// TIA Portal V19 export
FUNCTION_BLOCK "TYPIC_C105_IF_UPS"   // FB23, FBD
TITLE = TYPIC_C105_IF_UPS: No Break
{ S7_Optimized_Access := 'TRUE' }
AUTHOR : OCOTECH
FAMILY : Typical
NAME : C105.701
// Logisch Object Besturing: C105.601
// 
// De interne functie UPS verzorgt de bewaking van een Noobreak installatie.
// stored: MemoryReserve 10, SetENOAutomatically false
   VAR_INPUT
      IN_STS { ExternalAccessible := 'False'; ExternalVisible := 'False'; ExternalWritable := 'False'} : Bool;   // Status van UPS (Batterij / Werking / Bypass)
      IN_TYD { ExternalAccessible := 'False'; ExternalVisible := 'False'; ExternalWritable := 'False'} : Time;   // Resterende autonomietijd (min)
      IN_PWR { ExternalAccessible := 'False'; ExternalVisible := 'False'; ExternalWritable := 'False'} : Real;   // Resterend vermogen
      IN_SPA1 { ExternalAccessible := 'False'; ExternalVisible := 'False'; ExternalWritable := 'False'} : Real;   // Uitgangsspanning 1
      IN_SPA2 { ExternalAccessible := 'False'; ExternalVisible := 'False'; ExternalWritable := 'False'} : Real;   // Uitgangsspanning 2
      IN_SPA3 { ExternalAccessible := 'False'; ExternalVisible := 'False'; ExternalWritable := 'False'} : Real;   // Uitgangsspanning 3
      IN_STR1 { ExternalAccessible := 'False'; ExternalVisible := 'False'; ExternalWritable := 'False'} : Real;   // Uitgangsstroom 1
      IN_STR2 { ExternalAccessible := 'False'; ExternalVisible := 'False'; ExternalWritable := 'False'} : Real;   // Uitgangsstroom 2
      IN_STR3 { ExternalAccessible := 'False'; ExternalVisible := 'False'; ExternalWritable := 'False'} : Real;   // Uitgangsstroom 3
   END_VAR
   VAR_OUTPUT
      VAR_IF_UPS { ExternalAccessible := 'False'; ExternalVisible := 'False'; ExternalWritable := 'False'} : "C105_VAR_IF_UPS_TYPIC";   // Struct met alle variabelen naar bovenliggende functies
   END_VAR
   VAR
      STO { ExternalWritable := 'False'} : Struct   // Storingen
         A001 { ExternalAccessible := 'False'; ExternalVisible := 'False'} : Bool;   // No Break installatie in bypass
         A002 { ExternalAccessible := 'False'; ExternalVisible := 'False'} : Bool;   // No Break installatie uit bedrijf
      END_STRUCT;
      VAR { ExternalWritable := 'False'} : Struct   // Variabelen
         STS1 { ExternalAccessible := 'False'; ExternalVisible := 'False'} : Bool;   // Status UPS [In batterijwerking]
         STS2 { ExternalAccessible := 'False'; ExternalVisible := 'False'} : Bool;   // Status UPS [In bypass]
         STS3 { ExternalAccessible := 'False'; ExternalVisible := 'False'} : Bool;   // Status UPS [In normale werking]
         TYD { ExternalAccessible := 'False'; ExternalVisible := 'False'} : Time;   // Resterende autonomietijd [min]
         PWR { ExternalAccessible := 'False'; ExternalVisible := 'False'} : Real;   // Resterend vermogen
         SPA1 { ExternalAccessible := 'False'; ExternalVisible := 'False'} : Real;   // Uitgangsspanning 1
         SPA2 { ExternalAccessible := 'False'; ExternalVisible := 'False'} : Real;   // Uitgangsspanning 2
         SPA3 { ExternalAccessible := 'False'; ExternalVisible := 'False'} : Real;   // Uitgangsspanning 3
         STR1 { ExternalAccessible := 'False'; ExternalVisible := 'False'} : Real;   // Uitgangsstroom 1
         STR2 { ExternalAccessible := 'False'; ExternalVisible := 'False'} : Real;   // Uitgangsstroom 2
         STR3 { ExternalAccessible := 'False'; ExternalVisible := 'False'} : Real;   // Uitgangsstroom 3
      END_STRUCT;
   END_VAR
BEGIN

REGION Network 1: START
END_REGION

REGION Network 2: +++ Verwerking meetwaarden en statussen +++
   // De meetwaarde en status wordt ontvangen vanuit de interne sturing.
END_REGION

REGION Network 3: +++ Storingen +++
   // Storingen van het systeem
END_REGION

REGION Network 4: Storing A001: No Break installatie in bypass
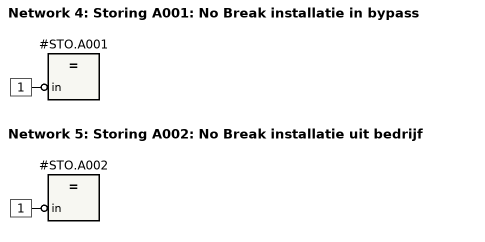
   #STO.A001 := NOT 1;
END_REGION

REGION Network 5: Storing A002: No Break installatie uit bedrijf
   #STO.A002 := NOT 1;
END_REGION

REGION Network 6 (SCL): EINDE
   // Variabelen van intern scada rakvlak naar outputs copieren
   #VAR_IF_UPS.STS1 := #VAR.STS1;
   #VAR_IF_UPS.STS2 := #VAR.STS2;
   #VAR_IF_UPS.STS3 := #VAR.STS3;
   #VAR_IF_UPS.TYD := #VAR.TYD;
   #VAR_IF_UPS.PWR := #VAR.PWR;
   #VAR_IF_UPS.SPA1 := #VAR.SPA1;
   #VAR_IF_UPS.SPA2 := #VAR.SPA2;
   #VAR_IF_UPS.SPA3 := #VAR.SPA3;
   #VAR_IF_UPS.STR1 := #VAR.STR1;
   #VAR_IF_UPS.STR2 := #VAR.STR2;
   #VAR_IF_UPS.STR3 := #VAR.STR3;
END_REGION
END_FUNCTION_BLOCK
